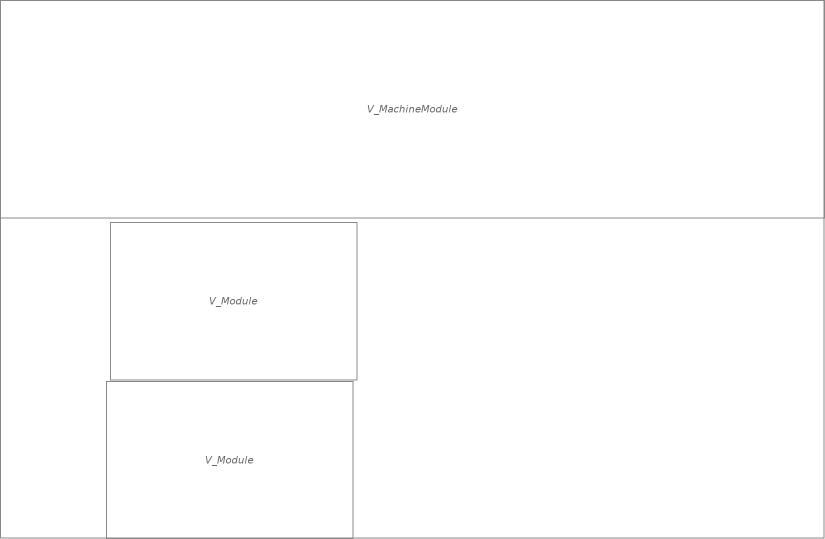
VISUALIZATION V_Application  // 825x539
    Frame (0,0 825x218)
        shows V_MachineModule(stVisu := MAIN.fbMyMachine.stPMLModuleBaseVISU)
    Frame (110,222 247x158)
        shows V_Module(stVisu := MAIN.fbMyMachine.fbEquipmentModule1.stPMLModuleBaseVISU)
    Frame (106,381 247x158)
        shows V_Module(stVisu := MAIN.fbMyMachine.fbEquipmentModule1.fb_EM1_ControlModule1.stPMLModuleBaseVISU)
END_VISUALIZATION

(* stored: Version 1.1.0.1, ProductVersion 3.1.4024.9
   Visu V_Application: Id {439e0c78-9d9c-4993-9985-93db18c60cfb} *)
